Fanuc KAREL source: kb00158.KL

-- PROVISIONAL review KL for V940-1; original PC SHA256 9c5432dc2ec5a54a35d097acf6a4486abf503e60246d8943adfb78902963c8ef
-- Incomplete behavior may be omitted. Consult companion uncertainty JSON. Do not deploy.
PROGRAM KB00158
%NOLOCKGROUP
BEGIN
  -- V9_ZERO_TABLE_METADATA_HINT layout=0002_ascii; no indexed target words; source/name/runtime held
  -- UNRESOLVED_PC offsets 5-12; opcodes 9D,23
  -- UNRESOLVED_PC offsets 17-24; opcodes 9D,23
  -- UNRESOLVED_PC offsets 29-45; opcodes 27,22,22,31
  -- UNRESOLVED_PC offsets 50-54; opcodes 7F
END KB00158
